ABB RAPID module: CircleMove.sys

MODULE CIRCLEMOVE(SYSMODULE, NOSTEPIN)
    PROC MoveCircle(
        robtarget pCenter,
        num Radius,
        speeddata Speed,
        zonedata Zone,
        PERS tooldata Tool\
        PERS wobjdata WObj)

            MoveCirecleImpl pCenter, Radius, Speed, Zone, Tool\
            WObj?WObj;

    ENDPROC
ENDMODULE
